Omron Sysmac Studio project AccumulationTimer_TP_Timer (Sysmac Studio 1.65.0.64007, StandardProject)

# Controller new_Controller_0: NX1P2-1040DT1 version 1.69
Task PrimaryTask (priority 4, period or condition 2000): Program0

VAR_GLOBAL
    BIO_Input_Bit_00 : BOOL;  (* at BuiltInIO://cpu/#0/Input_Bit_00 *)
    BIO_Input_Bit_01 : BOOL;  (* at BuiltInIO://cpu/#0/Input_Bit_01 *)
    BIO_Output_Bit_00 : BOOL;  (* at BuiltInIO://cpu/#0/Output_Bit_00 *)
    BIO_Output_Bit_01 : BOOL;  (* at BuiltInIO://cpu/#0/Output_Bit_01 *)
    IN_Start_Button : BOOL;
    INP : BOOL;
    StartButton : BOOL;
    StopButton : BOOL;
    Motor1 : BOOL;
    Motor2 : BOOL;
    AccumTimer1_Reset : BOOL;
    AccumTimer1_ET : TIME;
    Motor1_CalismaSuresi : INT;
    OUT_Motor1_Start : BOOL;
    OUT_Motor2_Start : BOOL;
    AccumTimer2_Reset : BOOL;
    AccumTimer2_ET : TIME;
    Motor2_CalismaSuresi : INT;
END_VAR
VAR_GLOBAL RETAIN
    E_TOF1_Saniye : INT;  (* published *)
    E_TON1_Saniye : INT;  (* published *)
END_VAR
VAR_GLOBAL
    TON1_ET : TIME;
    TOF1_ET : TIME;
    Actual_Time : DATE_AND_TIME;
    Time_Struct : _sDT;  (* Year UINT *)
    Equal : BOOL;
END_VAR

PROGRAM Program0
VAR
    Start : BOOL;
    AccumTimer1 : AccumulationTimer;
    AccumTimer2 : AccumulationTimer;
    TOF1 : TOF;
    TON1 : TOF;
END_VAR
VAR_EXTERNAL
    IN_Start_Button : BOOL;
    BIO_Output_Bit_00 : BOOL;
    INP : BOOL;
    BIO_Input_Bit_00 : BOOL;
    StartButton : BOOL;
    BIO_Input_Bit_01 : BOOL;
    StopButton : BOOL;
    Motor1 : BOOL;
    Motor2 : BOOL;
    BIO_Output_Bit_01 : BOOL;
    AccumTimer1_Reset : BOOL;
    AccumTimer1_ET : TIME;
    Motor1_CalismaSuresi : INT;
    OUT_Motor1_Start : BOOL;
    OUT_Motor2_Start : BOOL;
    AccumTimer2_Reset : BOOL;
    AccumTimer2_ET : TIME;
    Motor2_CalismaSuresi : INT;
    E_TOF1_Saniye : INT;
    E_TON1_Saniye : INT;
    TON1_ET : TIME;
    TOF1_ET : TIME;
    Actual_Time : DATE_AND_TIME;
    Time_Struct : _sDT;
    Equal : BOOL;
END_VAR

(* Section InOut: ladder, written here as Structured Text *)

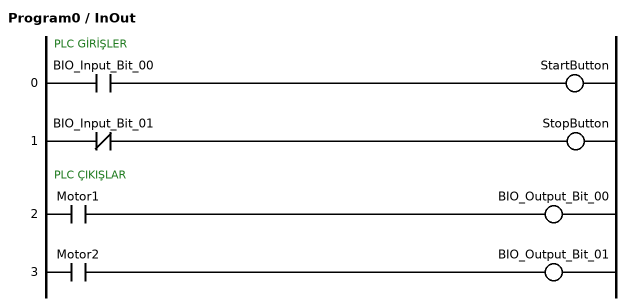
(* Rung 0: PLC GİRİŞLER *)
StartButton := BIO_Input_Bit_00;
(* Rung 1 *)
StopButton := NOT BIO_Input_Bit_01;
(* Rung 2: PLC ÇIKIŞLAR *)
BIO_Output_Bit_00 := Motor1;
(* Rung 3 *)
BIO_Output_Bit_01 := Motor2;

(* Section Multime_Ornek: ladder, written here as Structured Text *)

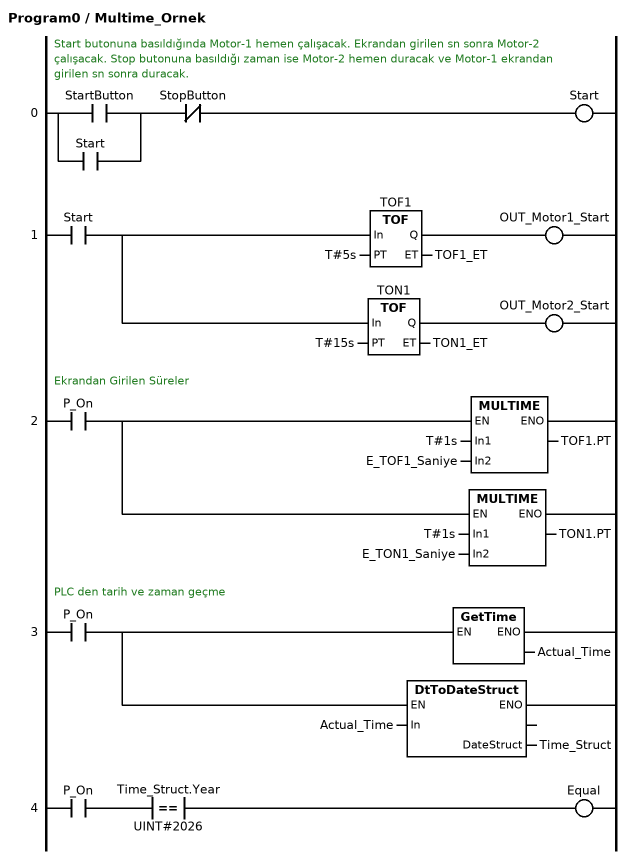
(* Rung 0: Start butonuna basıldığında Motor-1 hemen çalışacak. Ekrandan girilen sn sonra Motor-2 çalışacak. Stop butonuna basıldığı zaman ise Motor-2 hemen duracak ve Motor-1 ekrandan girilen sn sonra duracak. *)
Start := (StartButton OR Start) AND NOT StopButton;
(* Rung 1 *)
TOF1(In := Start, PT := T#5s, ET => TOF1_ET);
OUT_Motor1_Start := TOF1.Q;
TON1(In := Start, PT := T#15s, ET => TON1_ET);
OUT_Motor2_Start := TON1.Q;
(* Rung 2: Ekrandan Girilen Süreler *)
IF P_On THEN
    TOF1.PT := MULTIME(In1 := T#1s, In2 := E_TOF1_Saniye);
    TON1.PT := MULTIME(In1 := T#1s, In2 := E_TON1_Saniye);
END_IF;
(* Rung 3: PLC den tarih ve zaman geçme *)
IF P_On THEN Actual_Time := GetTime(); END_IF;
IF P_On THEN DtToDateStruct(In := Actual_Time, DateStruct => Time_Struct); END_IF;
(* Rung 4 *)
Equal := P_On AND (Time_Struct.Year = UINT#2026);
END_PROGRAM